Staubli VAL3: sum.pgx

public program sum(num& x_nInput[], num& x_nResult)
  local num l_nLength
  local num l_nElement
begin

  l_nLength = size(x_nInput)
  x_nResult = 0

  for l_nElement = 0 to l_nLength-1
    x_nResult = x_nResult + x_nInput[l_nElement]
  endFor

end
